{attribute 'qualified_only'}
{attribute 'strict'}
TYPE E_CommandDataState :
(
	Undefined := 0,
	CheckRequest,
	AddReservation,
	UpdateJobData,
	Done,
	Error
);
END_TYPE

(* stored: Version 1.1.0.1, ProductVersion 3.1.4024.5
   DUT E_CommandDataState: Id {fcf0416f-4b2b-4430-beb7-2f88c6326e5b} *)
